Staubli VAL3: sendTrajPtAck.pgx

public program sendTrajPtAck()
  local num l_nRetVal
begin
  // send message length (prefix)
  call sendData(siTcpIpMotion,rosTrajPtAck.prefix.nData,nInConnFlag)
  // send message header (msg type, comm type, reply code)
  call sendData(siTcpIpMotion,rosTrajPtAck.header.nData,nInConnFlag)
  call sendData(siTcpIpMotion,rosTrajPtAck.body.nData,nInConnFlag)
end
